// TIA Portal V19 export
DATA_BLOCK "M0940 G120_DI"   // DB940
VERSION : 0.0
// stored: AutoNumber false, InstanceOfName VSD Item Control, InstanceOfType FB
"VSD Item Control"
   // VAR_INPUT
   //    tripped : Bool;
   //    iso_On : Bool;
   //    maxTime : Int;
   //    rpm_Sp : Real := 0.0;
   //    hwID : HW_ANY;
   // END_VAR
   // VAR_IN_OUT
   //    output : Bool;
   //    ItemInfo : "ItemInfo_UDT";
   //    ItemTimer : "ItemTimer_UDT";
   //    ItemStatus : "ItemStatus_UDT";
   //    ItemCommand : "ItemCommand_UDT";
   // END_VAR
   // VAR
   //    vsd { S7_SetPoint := 'True'} : SinaSpeed;
   //    ActualSpeed : Real := 0.0;
   // END_VAR
BEGIN
END_DATA_BLOCK
